# EPICS substitutions: keithley2461App/Db/motor.substitutions
file "../../db/motor.db" {
  pattern
    {P,  M,  ADDR,  MRES,  DESC,  EGU}
    {alexHost:,  keithley2461Volt,  0,  "1e-7", "Voltage", "V"}
    {alexHost:,  keithley2461Curr,  1,  "1e-7", "Current", "A"}
}
